FUNCTION_BLOCK AE_AX_T_FF (* Toggle flip flop, bidirectional Socket (Toggle in, state back out via the same adapter) *)
  (* Standard: 61499-1 Annex A; Description: Copyright (c) 2026 HR Agrartechnik GmbH This program and the accompanying materials are made available under the terms of the Eclipse Public License 2.0 which is available at https://www.eclipse.org/legal/epl-2.0/ SPDX-License-Identifier: EPL-2.0 *)
  (* Version 1.0, 2026-09-03, Franz Höpfinger, HR Agrartechnik GmbH, wie AX_T_FF, aber mit bidirektionalem AE_AX-Socket statt plain CLK-EventInput + separatem AX-Plug - der Zustand geht ueber denselben Adapter zurueck *)
  PACKAGE adapter::events::bidirectional;
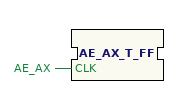
  SOCKETS
    CLK : adapter::types::bidirectional::AE_AX; (* Clock (in), Zustand (out) *)
  END_SOCKETS
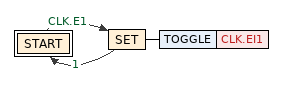
  EC_STATES
    START; (* Initial State *)
    SET : TOGGLE -> CLK.EI1; (* Initialization *)
  END_STATES
  EC_TRANSITIONS
    START TO SET := CLK.E1;
    SET TO START := 1;
  END_TRANSITIONS
  ALGORITHM TOGGLE IN ST:
CLK.DI1 := NOT CLK.DI1;
  END_ALGORITHM
END_FUNCTION_BLOCK
